// SIMATIC STEP 7 (V5.x) project S_Cizallado
// CPU: CPU312(1)
// station: P_ADR_BUS
// station: Hardware
// station: Equipo SIMATIC 300
// program: Programa S7(1)

SYMBOL_TABLE
"CONTADOR"	C 1	COUNTER
"CIZALLADO"	FB 2	FB 2	// Funcion que se encaga del cizallado de planchas
"CORTAR"	FC 1	FC 1	// Funcion de cortar las planchas
"BIT_DE_TRABAJO"	I 124.0	BOOL
"SENSOR"	I 124.1	BOOL
"SENSORABAJO"	I 124.2	BOOL
"SENSORARRIBA"	I 124.3	BOOL
"EXPULSADA"	I 124.4	BOOL
"START"	I 124.5	BOOL
"CARGAR_CONT"	I 124.6	BOOL
"Cycle Execution"	OB 1	OB 1
"PLANCHAS"	PIW 651	INT
"BAJARCUCHILLA"	Q 100.0	BOOL
"EXPULSARPLANCHA"	Q 100.1	BOOL
"BIT_OK"	Q 100.2	BOOL
"STBY"	Q 100.3	BOOL
END_SYMBOL_TABLE

FUNCTION_BLOCK "CIZALLADO"	// FB 2
TITLE = CIZALLADO
VERSION : 0.1
VAR_INPUT
  bit_de_trabajo : BOOL ;
  SENSOR : BOOL ;
  PLANCHAS : INT ;
  SENSORABAJO : BOOL ;
  SENSORARRIBA : BOOL ;
  EXPULSADA : BOOL ;
  CONTADOR : COUNTER ;
  START : BOOL ;
END_VAR
VAR_OUTPUT
  BAJARCUCHILLA : BOOL ;
  EXPULSARPLANCHA : BOOL ;
  STBY : BOOL ;
  BIT_OK : BOOL ;
END_VAR
VAR
  X41 : BOOL ;
  M3 : BOOL ;
  X43 : BOOL ;
  FP_BDT : BOOL ;
  FP_START : BOOL ;
  INICORTAR : BOOL ;
  S2 : BOOL ;
  BDT_CORTAR : BOOL ;
  OK_CORTAR : BOOL ;
  STBY_CORTAR : BOOL ;
  CORTADO : BOOL ;
END_VAR
BEGIN
NETWORK
TITLE = Arranque
      A     #bit_de_trabajo;
      FP    #FP_BDT;
      =     #BDT_CORTAR;
      S     #X41;
      R     #M3;
      R     #X43;
      R     #INICORTAR;
      R     #CORTADO;
      R     #BIT_OK;
      R     #S2;
NETWORK
TITLE = De x41 a M3
      A     #X41;
      A     #SENSOR;
      A     #STBY_CORTAR;
      A     #START;
      FP    #FP_START;
      R     #X41;
      S     #M3;
NETWORK
TITLE = De M3 a x43
      A     #M3;
      A     #CORTADO;
      R     #M3;
      S     #X43;
NETWORK
TITLE = de x43 a x41
      A     #X43;
      T     LD 0;
      TAK;
      T     LD 4;
      L     #CONTADOR;
      T     LW 8;
      L     LD 4;
      L     LD 0;
      AN    C [LW 8];
      R     #X43;
      S     #S2;
NETWORK
TITLE = de x43 a X41
      A     #X43;
      T     LD 0;
      TAK;
      T     LD 4;
      L     #CONTADOR;
      T     LW 8;
      L     LD 4;
      L     LD 0;
      A     C [LW 8];
      R     #X43;
      S     #X41;
NETWORK
TITLE = De M3 a x43 con call M3
      CALL  "CORTAR" (
           bit_de_trabajo           := #BDT_CORTAR,
           SENSORABAJO              := #SENSORABAJO,
           SENSORARRIBA             := #SENSORARRIBA,
           EXPULSADA                := #EXPULSADA,
           START                    := #INICORTAR,
           OK                       := #OK_CORTAR,
           BAJARCUCHILLA            := #BAJARCUCHILLA,
           EXPULSARPLANCHA          := #EXPULSARPLANCHA,
           bit_ok                   := #CORTADO,
           STBY                     := #STBY_CORTAR);
NETWORK
TITLE =
      A     #M3;
      A     #CORTADO;
      R     #M3;
      S     #X43;
NETWORK
TITLE =
      A     #M3;
      =     #INICORTAR;
NETWORK
TITLE = Cuenta el numero de planchas cortadas
      A     #X43;
      =     #OK_CORTAR;
      T     LD 0;
      TAK;
      T     LD 4;
      L     #CONTADOR;
      T     LW 8;
      L     LD 4;
      L     LD 0;
      CD    C [LW 8];
NETWORK
TITLE =
      A     #X41;
      =     #STBY;
NETWORK
TITLE =
      A     #S2;
      =     #BIT_OK;
END_FUNCTION_BLOCK

FUNCTION "CORTAR" : VOID	// FC 1
TITLE = CORTAR
VERSION : 0.1
VAR_INPUT
  bit_de_trabajo : BOOL ;
  SENSORABAJO : BOOL ;
  SENSORARRIBA : BOOL ;
  EXPULSADA : BOOL ;
  START : BOOL ;
  OK : BOOL ;
END_VAR
VAR_OUTPUT
  BAJARCUCHILLA : BOOL ;
  EXPULSARPLANCHA : BOOL ;
  bit_ok : BOOL ;
  STBY : BOOL ;
END_VAR
VAR_TEMP
  x51 : BOOL ;
  x52 : BOOL ;
  x53 : BOOL ;
  s3 : BOOL ;
  FP_BDT : BOOL ;
  X50 : BOOL ;
  FP_START : BOOL ;
END_VAR
BEGIN
NETWORK
TITLE = Arranque
      A     #bit_de_trabajo;
      FP    #FP_BDT;
      S     #X50;
      R     #x51;
      R     #x52;
      R     #x53;
      R     #s3;
NETWORK
TITLE = de x51 a x52
      A     #x51;
      A     #SENSORABAJO;
      R     #x51;
      S     #x52;
NETWORK
TITLE = de x52 a x53
      A     #x52;
      A     #SENSORARRIBA;
      R     #x52;
      S     #x53;
NETWORK
TITLE = de x53 a s3
      A     #x53;
      A     #EXPULSADA;
      R     #x53;
      S     #s3;
NETWORK
TITLE = Accion x51
      A     #x51;
      =     #BAJARCUCHILLA;
NETWORK
TITLE = Accion x53
      A     #x53;
      =     #EXPULSARPLANCHA;
NETWORK
TITLE = Accion final
      A     #s3;
      =     #bit_ok;
NETWORK
TITLE =
      A     #s3;
      A     #OK;
      R     #s3;
      S     #X50;
NETWORK
TITLE =
      A     #X50;
      A     #START;
      FP    #FP_START;
      R     #X50;
      S     #x51;
NETWORK
TITLE =
      A     #X50;
      =     #STBY;
END_FUNCTION

DATA_BLOCK DB 1
VERSION : 0.0
"CIZALLADO"
BEGIN
END_DATA_BLOCK

ORGANIZATION_BLOCK "Cycle Execution"	// OB 1
TITLE = "Main Program Sweep (Cycle)"
VERSION : 0.1
VAR_TEMP
  OB1_EV_CLASS : BYTE ;	//Bits 0-3 = 1 (Coming event), Bits 4-7 = 1 (Event class 1)
  OB1_SCAN_1 : BYTE ;	//1 (Cold restart scan 1 of OB 1), 3 (Scan 2-n of OB 1)
  OB1_PRIORITY : BYTE ;	//Priority of OB Execution
  OB1_OB_NUMBR : BYTE ;	//1 (Organization block 1, OB1)
  OB1_RESERVED_1 : BYTE ;	//Reserved for system
  OB1_RESERVED_2 : BYTE ;	//Reserved for system
  OB1_PREV_CYCLE : INT ;	//Cycle time of previous OB1 scan (milliseconds)
  OB1_MIN_CYCLE : INT ;	//Minimum cycle time of OB1 (milliseconds)
  OB1_MAX_CYCLE : INT ;	//Maximum cycle time of OB1 (milliseconds)
  OB1_DATE_TIME : DATE_AND_TIME ;	//Date and time OB1 started
END_VAR
BEGIN
NETWORK
TITLE =
      CALL  "CIZALLADO" , DB 1 (
           bit_de_trabajo           := "BIT_DE_TRABAJO",
           SENSOR                   := "SENSOR",
           PLANCHAS                 := "PLANCHAS",
           SENSORABAJO              := "SENSORABAJO",
           SENSORARRIBA             := "SENSORARRIBA",
           EXPULSADA                := "EXPULSADA",
           CONTADOR                 := "CONTADOR",
           START                    := "START",
           BAJARCUCHILLA            := "BAJARCUCHILLA",
           EXPULSARPLANCHA          := "EXPULSARPLANCHA",
           STBY                     := "STBY",
           BIT_OK                   := "BIT_OK");
NETWORK
TITLE =
      A     "CARGAR_CONT";
      L     "PLANCHAS";
      S     "CONTADOR";
END_ORGANIZATION_BLOCK
